FUNCTION_BLOCK machineStation EXTENDS stateMachine
VAR_INPUT
	
	ioImage      : machineImage;

END_VAR
VAR
	
	activeState 	: machineStates;
	
	resetTime   	: TIME := T#2S;           // Време за ресет след ативиране на EMG stop
	resetSig		: BOOL := FALSE; 
	resetTimer		: TON;
	commandReady	: BOOL; 				  // Има приета нова команда
	errorPuls 		: R_TRIG;			      // Има нова грешка в машината
	
	purgeIndexDone  : BOOL := FALSE; 		  // Изчаква да се извадят всички бройки от масата
	purgeRobotDone  : BOOL := FALSE; 		  // Робота е приключил работа
	purgeStackers   : BOOL := FALSE;          // Стакерите са извадили всички тари от тях
	
	startZumer			   : BOOL;									   // Упр. на сигнален зумер
	zumerTimer1			   : TON;
	zumerTimer2			   : TON;
	zumerTimer3			   : TON;
	zumerBeep			   : INT;

END_VAR
VAR // added by the converter: edge detectors and wires of the graphical bodies
    _w1, _w2, _w3 : BOOL;
END_VAR


// Има разлики спрямо останалите станций на машита
// Някой states липсват и не може тази станция да минава в stop режим

zumer();                  // Упр. на сигният зумер

// Сигнали за HMI

	TagsHMI.activeEmg       := io.getX(ioImage.xEmgBnt);
	TagsHMI.doorsOpen       := io.getX(ioImage.xDoors);         
	TagsHMI.noAir           := io.getX(ioImage.xAirOk);            
	TagsHMI.robotEmgActive  := io.getX(ioImage.xRobotEmgOk);            
	TagsHMI.robotNoCom      := TagsRobot.robotComOnline;    
	TagsHMI.robotError      := TagsRobot.robotError;    


errorPuls(CLK := Global.machError); 

IF NOT io.getX(ioImage.xDoors) AND io.getX(ioImage.xAirOk) AND io.getX(ioImage.xEmgBnt) THEN
	Global.openDoors := TRUE;						// Има отворена вратa
	Global.emgStop   := FALSE;
	setDisplayState(machineDisplayStates.dStOpenDoors);
	setEmg(emgOrAlarm := TRUE);
	
ELSIF NOT io.getX(ioImage.xEmgBnt) THEN
	Global.emgStop   := TRUE; 					   //  Авариен стоп
	Global.openDoors := FALSE;	
	setDisplayState(machineDisplayStates.dStEMGButtonDown);
	setEmg(emgOrAlarm := TRUE);
	
ELSIF NOT io.getX(ioImage.xAirOk)  THEN
 	Global.emgStop   := TRUE; 					   // Няма оперативно налягане на въздуха   
	Global.openDoors := FALSE;	
	setDisplayState(machineDisplayStates.dStNoAirSupplay);
	setEmg(emgOrAlarm := TRUE);	
	
END_IF

IF NOT io.getX(ioImage.xRobotEmgOk) AND TagsRobot.robotComOnline THEN
 	Global.emgStop   := TRUE; 	                   //  Авариен стоп  на робота
	Global.RobotEMG  := TRUE;				      
	setDisplayState(machineDisplayStates.dStMachineRobotEMG);
	setEmg(emgOrAlarm := TRUE);	
	
ELSIF io.getX(ioImage.xRobotEmgOk) AND NOT TagsRobot.robotComOnline THEN
 	Global.emgStop     := TRUE; 	               //  Липса на комуникация с робота
	Global.RobotNoCom  := TRUE;				      
	setDisplayState(machineDisplayStates.dStMachineRobotNoCom);
	setEmg(emgOrAlarm := TRUE);		
END_IF

IF errorPuls.Q THEN
	setEmg(emgOrAlarm := FALSE);	
	Global.startZumer := TRUE;
END_IF

setStateVars(ioImage, activeState);


CASE activeState OF 
	
//  *** Start Up
//  Старт на станцията след подаване на захр.

	machineStates.stStartUp:
		Global.emgStop       := FALSE;
		Global.openDoors     := FALSE;
		Global.emgStopSignal := FALSE;
		resetSig             := FALSE;
		commandReady         := FALSE;
		purgeIndexDone       := FALSE;
		purgeRobotDone       := FALSE;
		purgeStackers		 := FALSE;
		Global.commands      := controlCommands.null;
		setDisplayState(machineDisplayStates.dStStartUp);
		NextState(machineStates.stInit);
	
//  *** Safety stop 
//  Има отворена врата, няма въздух или има натисната губа
//  Към всички станций се подава EMG сигнал

	machineStates.stSafetyStop:
		Global.commands      := controlCommands.null;
		Global.emgStopSignal := TRUE;
		resetTimer(IN := resetSig, PT := resetTime);
		
		IF      io.getX(ioImage.xDoors) 
			AND io.getX(ioImage.xAirOk) 
			AND io.getX(ioImage.xEmgBnt) 
			AND io.getX(ioImage.xRobotEmgOk)
            AND TagsRobot.robotComOnline  THEN
				resetSig := TRUE;
				IF resetTimer.Q THEN	
					resetSig      := FALSE;
					nextState(machineStates.stInit);
				END_IF
		END_IF	

//  *** Init 
//  Инициализация на всички станций 
			
	machineStates.stInit:
		setDisplayState(machineDisplayStates.dStMachineStandBy);
		
		CASE Global.commands OF	
			controlCommands.start, 
			controlCommands.stop:
		        commandReady         := TRUE;
				Global.machError     := FALSE;
			    Global.emgStopSignal := FALSE;
			    nextState(machineStates.stReady);
				
			    Stations.incCommStBase.DoInit      := TRUE;			
			    Stations.sLoadStBase.DoInit        := TRUE;
				Stations.sUnloadStBase.DoInit      := TRUE;
				Stations.insertLoadStBase.DoInit   := TRUE;
				Stations.insertUnloadStBase.DoInit := TRUE;				
				Stations.roboStBase.DoInit         := TRUE;		
			
		END_CASE

// *** Ready 
// Синхронизира всички станций след подаване на захранването

	machineStates.stReady:
		depSync(Stations.incCommStBase,      globalDeps.depIncCommModeDone); 
		depSync(Stations.sLoadStBase,        globalDeps.depSLoadInit);
		depSync(Stations.sUnloadStBase,      globalDeps.depSUnloadInit);
		depSync(Stations.insertLoadStBase,   globalDeps.depILoadInitDone);
		depSync(Stations.insertUnloadStBase, globalDeps.depULoadInitDone);
		depSync(Stations.roboStBase,         globalDeps.depRoboInitDone);	
	
		nextState(machineStates.stCheckState);	
		
// *** Check state 
// В зависимост от зададената команда се задава следващо състояние

	machineStates.stCheckState:	
		IF NOT Global.purgeActive THEN	
			
			CASE Global.commands OF	
				controlCommands.start:
					nextState(machineStates.stAutoRun);
		   		controlCommands.stop:		
					nextState(machineStates.stStopping);
			END_CASE
			
		ELSE
			// Активна е purge процедура
			// Изчаква да се изпразни масата
			IF NOT purgeIndexDone THEN
				nextState(machineStates.stPurgeDialIndexSync);
			END_IF
			
			// Изчаква робота на приключи работа
			IF NOT purgeRobotDone THEN
				nextState(machineStates.stPurgeRobot);
			END_IF		

			// Изчаква стакерите да изкарат тарите в тях
			IF NOT purgeStackers THEN
				nextState(machineStates.stPurgeStackers);
			END_IF	
			
			nextState(machineStates.stPurgeDone);
			
		END_IF	

//  *** Stopping
//  Изчакват се всички станций да спрат

	machineStates.stStopping:
		setDisplayState(machineDisplayStates.dStMachineIsStopping);
		depSignal(globalDeps.depMachineStopping);
		depSync(Stations.incCommStBase,      globalDeps.depIncStop);		
		depSync(Stations.sLoadStBase,        globalDeps.depSLoadStop);
		depSync(Stations.sUnloadStBase,      globalDeps.depSUnloadStop);
		depSync(Stations.insertLoadStBase,   globalDeps.depILoadStop);
		depSync(Stations.insertUnloadStBase, globalDeps.depULoadStop);
		depSync(Stations.roboStBase,         globalDeps.depRoboStop);
		
		nextState(machineStates.stStopMach);
		
//  *** Stop 
//  Машината е спряна

	machineStates.stStopMach:	
		IF commandReady THEN
			Global.commands    := controlCommands.null;
			commandReady       := FALSE;	
		END_IF
	    setDisplayState(machineDisplayStates.dStMachineIsStopped);
	  
	    CASE Global.commands OF	
	      controlCommands.start:
		  	 commandReady := TRUE;
			 IF NOT Global.purgeActive THEN
		  		 nextState(machineStates.stAutoRun);	
			 ELSE
		  		 nextState(machineStates.stPurgeStart);
			 END_IF				 
							
		END_CASE	
	  
//  *** Auto run
//  Автоматичен режим

	machineStates.stAutoRun:
		IF commandReady THEN
			Global.commands    := controlCommands.null;
	    	commandReady       := FALSE;	
		END_IF
	    setDisplayState(machineDisplayStates.dStAutoRun);
		depSignal(globalDeps.depMachineAuto);
		IF Global.commands = controlCommands.stop THEN
		  	 commandReady := TRUE;				
		  	 nextState(machineStates.stStopping);			
		END_IF

// *** Purge - Start
// Изчистване на останалите в машита бройките
	
	machineStates.stPurgeStart:
		purgeIndexDone       := FALSE;
		purgeRobotDone       := FALSE;
		purgeStackers		 := FALSE;
		setDisplayState(machineDisplayStates.dStMachinePurgeActive);
		depSignal(globalDeps.depMachinePurgeStart);
		nextState(machineStates.stPurgeDialIndexSync);	
		
// *** Purge - Dial Index Sync
// Изчаква масата на InC да се завърти колкое необходимо пъти
// зада се изчистят останалите броки от нея
	
	machineStates.stPurgeDialIndexSync:	
		purgeIndexDone := FALSE;
		depSync(Stations.incCommStBase, globalDeps.depIncPurgeDone);
		nextState(machineStates.stPurgeRobot);		
		
// *** Purge - Robot Start
// Команда purge към робота
	
	machineStates.stPurgeRobot:	
		purgeIndexDone := TRUE;
		purgeRobotDone := FALSE;
		depSignal(globalDeps.depMachinePurgeRobot);
		depSync(Stations.roboStBase, globalDeps.depRoboPurgeDone);
		nextState(machineStates.stPurgeStackers);
		
// *** Purge - Stackers
// Команда purge към стакерите
	
	machineStates.stPurgeStackers:
		purgeRobotDone := TRUE;
		purgeStackers  := FALSE;	
		depSignal(globalDeps.depMacinePurgeStackers);	
		depSync(Stations.sLoadStBase,   globalDeps.depSLoadPurgeDone);	
		depSync(Stations.sUnloadStBase, globalDeps.depSUnloadPurgeDone);	
		nextState(machineStates.stPurgeDone);

// *** Purge - Done

	machineStates.stPurgeDone:	
		purgeStackers		 := TRUE;
		Global.purgeActive   := FALSE;
	    TagsHMI.startPurge   := FALSE;		
		nextState(machineStates.stStop);				
	
//  *** Machine error
//  В някоя станция има грешка

	machineStates.stMachError:
		Global.commands    := controlCommands.null;
		setDisplayState(machineDisplayStates.dStStationError);		
	
END_CASE

METHOD PRIVATE setEmg
VAR_INPUT
	
	emgOrAlarm				: Bool; 				// Дали метода е извикам за EMG stop или аларма

END_VAR

// Когато има EMG ситуация или аларма, се задава съответният state, 
// без оглед на текущото състояние на state машината.
// Аварийното спиратен е с по-голям приоритет от алармата

	stBase.DependencyState       := Consts.NO_DEPENDENCY;
	depActive                    := FALSE;
	syncActive                   := FALSE;
	statePass 			   		 := FALSE;
	depCount                     := 0;
	MEMSET(ADR(syncArr), 0, SIZEOF(syncArr));
	
	IF emgOrAlarm THEN
		stCurrentState               := machineStates.stSafetyStop;
		stBase.CurrentState          := machineStates.stSafetyStop;
	ELSE
		stCurrentState               := machineStates.stMachError;
		stBase.CurrentState          := machineStates.stMachError;
	END_IF
END_METHOD

ACTION zumer:
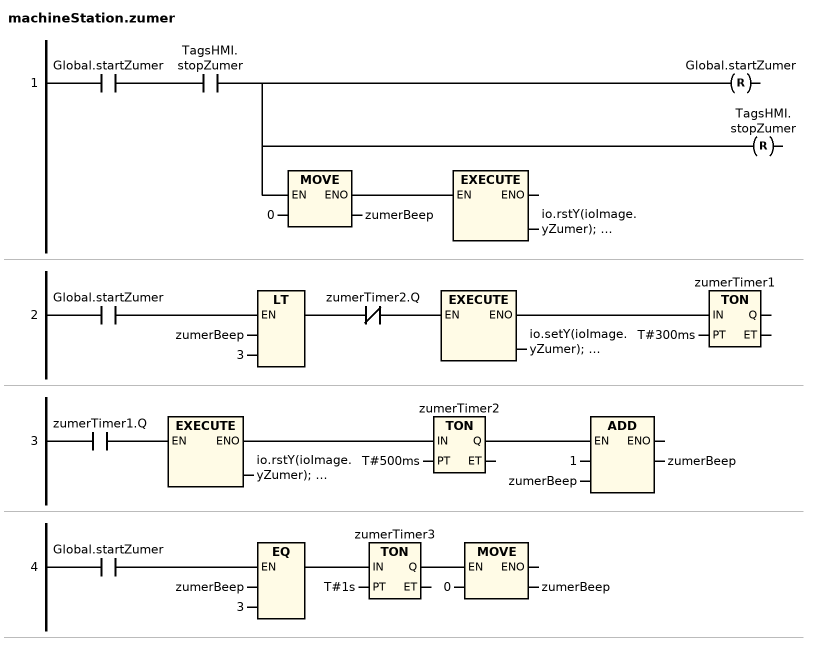
// NETWORK 1
_w1 := Global.startZumer AND TagsHMI.stopZumer;
Global.startZumer R= _w1;
TagsHMI.stopZumer R= _w1;
IF _w1 THEN zumerBeep := 0; END_IF
IF _w1 THEN io.rstY(ioImage.yZumer); END_IF

// NETWORK 2
_w2 := (Global.startZumer AND zumerBeep < 3) AND NOT zumerTimer2.Q;
IF _w2 THEN io.setY(ioImage.yZumer); END_IF
zumerTimer1(IN := _w2, PT := T#300ms); // TON

// NETWORK 3
_w3 := zumerTimer1.Q;
IF _w3 THEN io.rstY(ioImage.yZumer); END_IF
zumerTimer2(IN := _w3, PT := T#500ms); // TON
IF zumerTimer2.Q THEN zumerBeep := 1 + zumerBeep; END_IF

// NETWORK 4
zumerTimer3(IN := Global.startZumer AND zumerBeep = 3, PT := T#1s); // TON
IF zumerTimer3.Q THEN zumerBeep := 0; END_IF
END_ACTION

END_FUNCTION_BLOCK

(* stored: Version 1.1.0.1, ProductVersion 3.1.4024.3
   POU machineStation: Id {4c5bfae4-5dc2-4ad0-b7cc-a8d6904ca8f2}, SpecialFunc None
   Method setEmg: Id {2a2162a7-19cb-4fac-b41b-b6f7af5ee9a4}
   Action zumer: Id {386b5956-aed7-4313-9bb0-811f93e676e4} *)
